// TIA Portal V20 export
VAR_GLOBAL   // PLC tag table "LKinCtrl_HMI_Editor"
END_VAR
VAR_GLOBAL CONSTANT   // user constants
   LKINCTRL_NO_OF_PATH_UNDOS_PATH_EDITOR : Int := 10;   // Total number of undos for changes in path table.
   LKINCTRL_NO_OF_POINT_UNDOS_POINT_EDITOR : Int := 10;   // Total number of undos in the point editor.
   LKINCTRL_NO_OF_COMMAND_UNDOS_PATH_EDITOR : Int := 30;   // Total number of undos for changes in command editor.
END_VAR
